VAR
	alarmP1trig: RS;		(*Триггер - защелка аварии насоса 1.*)
	alarmP2trig: RS;		(*Триггер - защелка аварии насоса 2.*)
	stopPump1Detector: F_TRIG;		(*Детектор спада сигнала (останов) насоса 1.*)
	stopPump2Detector: F_TRIG;		(*Детектор спада сигнала (останов) насоса 2.*)
	delayAfterStopP2: TOF;		(*Таймер задержки на включение
насоса 1 после останова насоса 2.*)
	delayAfterStopP1: TOF;		(*Таймер задержки на включение
насоса 2 после останова насоса 1.*)
	antiFreqStartPump1: TOF;		(*Таймер - предохранитель от частых пусков насоса 1.*)
	antiFreqStartPump2: TOF;		(*Таймер - предохранитель от частых пусков насоса 2.*)
	startPump1Trig: RS;		(*RS триггер на пуск насоса 1.*)
	startPump2Trig: RS;		(*RS триггер на пуск насоса 2.*)
	stopPump1: F_TRIG;		(*Сигнал на останов насоса 1.*)
	stopPump2: F_TRIG;		(*Сигнал на останов насоса 2.*)
END_VAR
VAR_INPUT
	startP1: BOOL;		(*Сигнал на запуск насоса 1.
Активен - пуск, неактивен - стоп.*)
	startP2: BOOL;		(*Сигнал на запуск насоса 2.
Активен - пуск, неактивен - стоп.*)
	alarmP1input: BOOL;		(*Сигнал авария от насоса 1.*)
	alarmP2input: BOOL;		(*Сигнал авария от насоса 2.*)
	stop: BOOL;		(*Сигнал на останов. Пока активен - пусков нет.
Общий на оба насоса.*)
	reset: BOOL;		(*Сброс аварий.*)
	delayTime: WORD := 300;		(*Задержка на повторный пуск в секундах.
Если ко входу ничего не подключено, то 300сек.*)
END_VAR
VAR_OUTPUT
	pump1on: BOOL;		(*Выход на запуск насоса 1.*)
	pump2on: BOOL;		(*Выход на запуск насоса 2.*)
	nextStartP1Timer: WORD;		(*Счетчик секунд до возможности повторного пуска насоса 1.*)
	nextStartP2Timer: WORD;		(*Счетчик секунд до возможности повторного пуска насоса 2.*)
	alarmP1: BOOL;		(*Статус - авария насоса 1.*)
	alarmP2: BOOL;		(*Статус - авария насоса 2.*)
END_VAR
VAR (* helpers for the ST form of the networks *)
	_t203 : TIME;
END_VAR
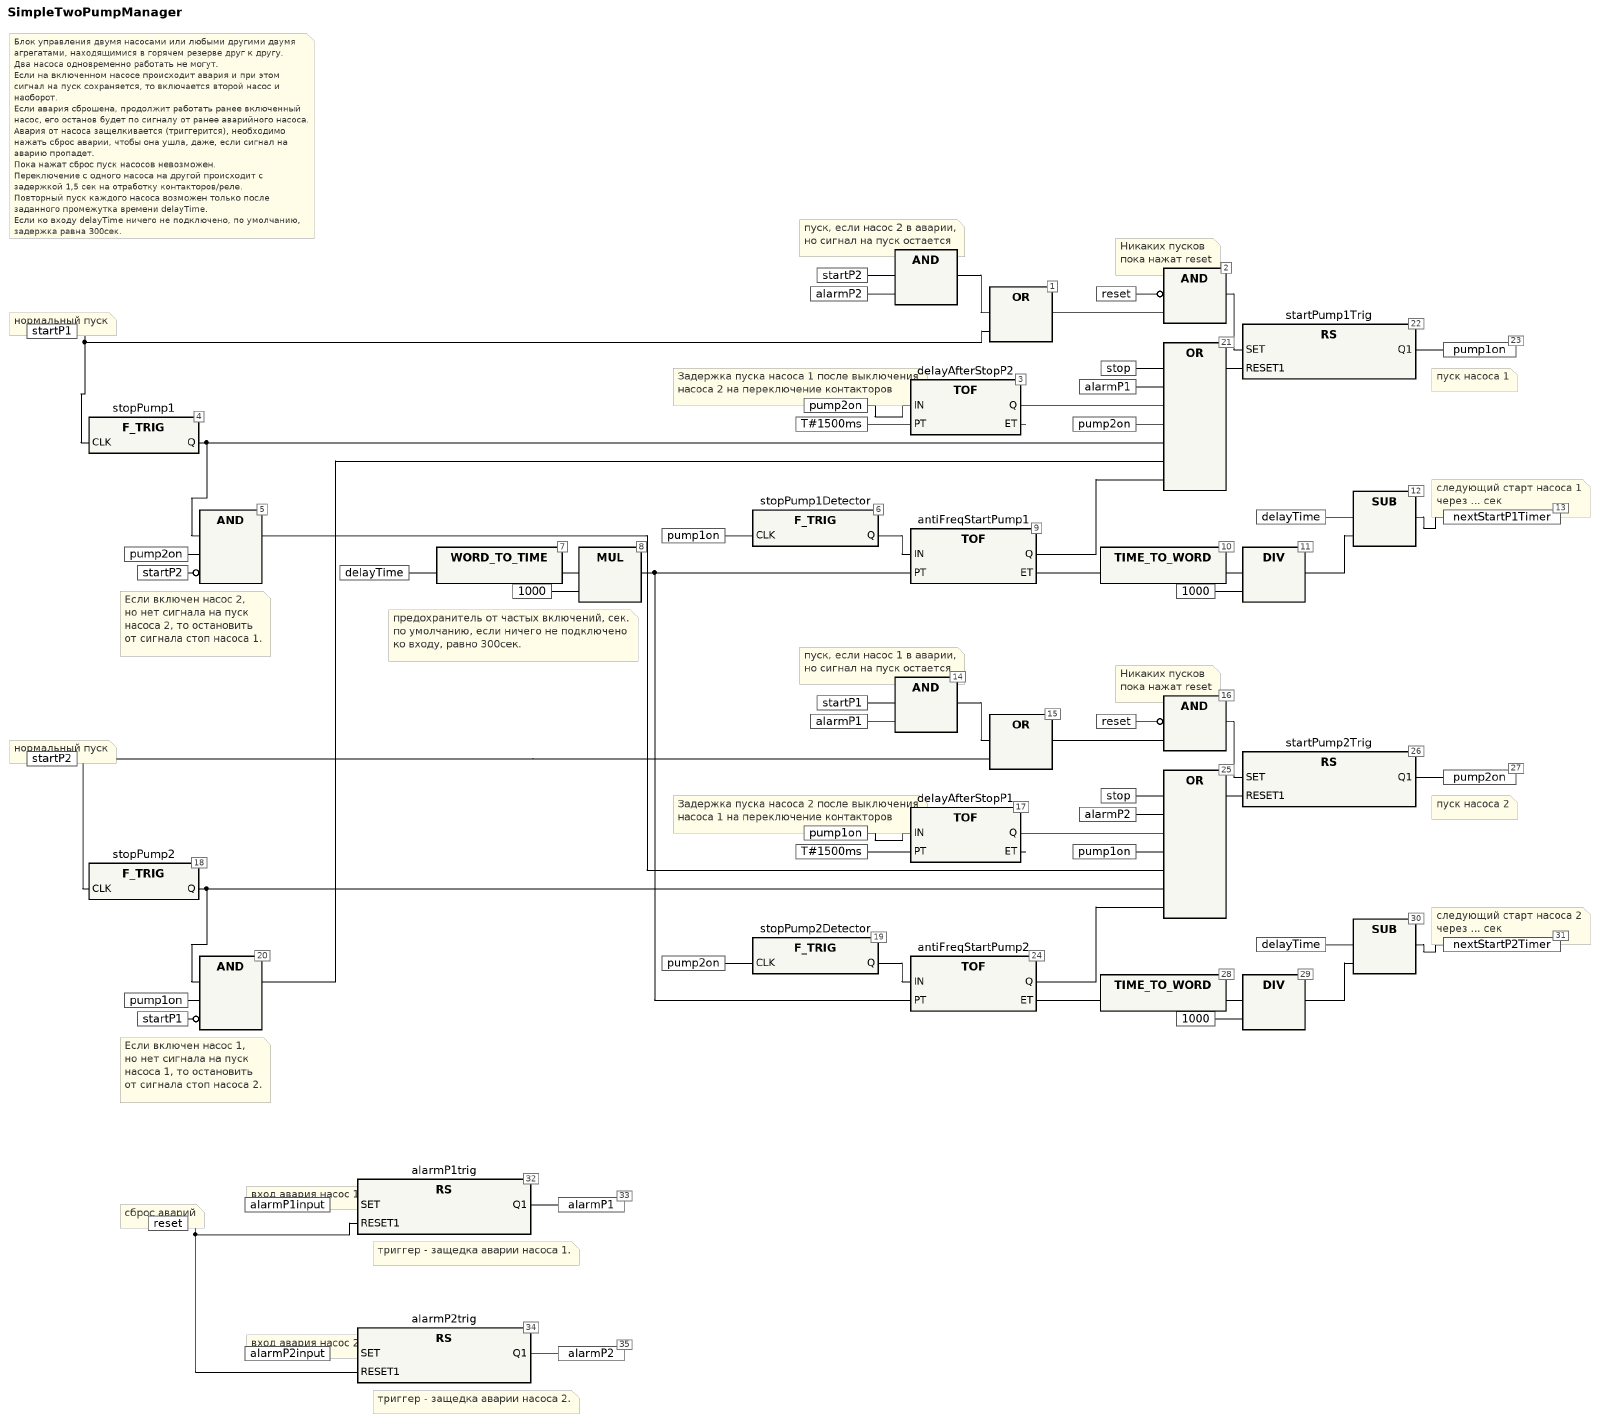
[picture p13: SimpleTwoPumpManager (CFC)]
_CFC_ (* Continuous Function Chart, elements in execution order *)
(* Задержка пуска насоса 2 после выключения / насоса 1 на переключение контакторов *)
(* cледующий старт насоса 2 / через ... сек *)
(* триггер - защедка аварии насоса 2. *)
(* cледующий старт насоса 1 / через ... сек *)
(* триггер - защедка аварии насоса 1. *)
(* предохранитель от частых включений, сек. / по умолчанию, если ничего не подключено / ко входу, равно 300сек. *)
(* пуск, если насос 1 в аварии, / но сигнал на пуск остается *)
(* нормальный пуск *)
(* пуск, если насос 2 в аварии, / но сигнал на пуск остается *)
(* нормальный пуск *)
(* Задержка пуска насоса 1 после выключения / насоса 2 на переключение контакторов *)
(* вход авария насос 1 *)
(* сброс аварий *)
(* пуск насоса 1 *)
(* вход авария насос 2 *)
(* пуск насоса 2 *)
(* Блок управления двумя насосами или любыми другими двумя агрегатами, находящимися в горячем резерве друг к другу. / Два насоса одновременно работать не могут. / Если на включенном насосе происходит авария и при этом сигнал на пуск сохраняется, то включается второй насос и наоборот. / Если авария сброшена, продолжит работать ранее включенный насос, его останов будет по сигналу от ранее аварийного насоса. / Авария от насоса защелкивается (триггерится), необходимо нажать сброс аварии, чтобы она ушла, даже, если сигнал на аварию пропадет. / Пока нажат сброс пуск насосов невозможен. / Переключение с одного насоса на другой происходит с задержкой 1,5 сек на отработку контакторов/реле. / Повторный пуск каждого насоса возможен только после заданного промежутка времени delayTime. / Если ко входу delayTime ничего не подключено, по умолчанию, задержка равна 300сек. *)
(* Никаких пусков / пока нажат reset *)
(* Никаких пусков / пока нажат reset *)
(* Если включен насос 2, / но нет сигнала на пуск / насоса 2, то остановить / от сигнала стоп насоса 1. *)
(* Если включен насос 1, / но нет сигнала на пуск / насоса 1, то остановить / от сигнала стоп насоса 2. *)
#0 AND(startP2, alarmP2)
#1 OR(#0, startP1)
#2 AND(NOT reset, #1)
#3 delayAfterStopP2:TOF(IN: pump2on, PT: T#1500ms)
#4 stopPump1:F_TRIG(CLK: startP1)
#5 AND(#4.Q, pump2on, NOT startP2)
#6 stopPump1Detector:F_TRIG(CLK: pump1on)
#7 WORD_TO_TIME(delayTime)
#8 MUL(#7, 1000)
#9 antiFreqStartPump1:TOF(IN: #6.Q, PT: #8)
#10 TIME_TO_WORD(#9.ET)
#11 DIV(#10, 1000)
#12 SUB(delayTime, #11)
#13 nextStartP1Timer <= #12
#14 AND(startP1, alarmP1)
#15 OR(#14, startP2)
#16 AND(NOT reset, #15)
#17 delayAfterStopP1:TOF(IN: pump1on, PT: T#1500ms)
#18 stopPump2:F_TRIG(CLK: startP2)
#19 stopPump2Detector:F_TRIG(CLK: pump2on)
#20 AND(#18.Q, pump1on, NOT startP1)
#21 OR(stop, alarmP1, #3.Q, pump2on, #4.Q, #20, #9.Q)
#22 startPump1Trig:RS(SET: #2, RESET1: #21)
#23 pump1on <= #22.Q1
#24 antiFreqStartPump2:TOF(IN: #19.Q, PT: #8)
#25 OR(stop, alarmP2, #17.Q, pump1on, #5, #18.Q, #24.Q)
#26 startPump2Trig:RS(SET: #16, RESET1: #25)
#27 pump2on <= #26.Q1
#28 TIME_TO_WORD(#24.ET)
#29 DIV(#28, 1000)
#30 SUB(delayTime, #29)
#31 nextStartP2Timer <= #30
#32 alarmP1trig:RS(SET: alarmP1input, RESET1: reset)
#33 alarmP1 <= #32.Q1
#34 alarmP2trig:RS(SET: alarmP2input, RESET1: reset)
#35 alarmP2 <= #34.Q1
_END_CFC_
(* the same logic as Structured Text *)
(* Задержка пуска насоса 2 после выключения / насоса 1 на переключение контакторов *)
(* cледующий старт насоса 2 / через ... сек *)
(* триггер - защедка аварии насоса 2. *)
(* cледующий старт насоса 1 / через ... сек *)
(* триггер - защедка аварии насоса 1. *)
(* предохранитель от частых включений, сек. / по умолчанию, если ничего не подключено / ко входу, равно 300сек. *)
(* пуск, если насос 1 в аварии, / но сигнал на пуск остается *)
(* нормальный пуск *)
(* пуск, если насос 2 в аварии, / но сигнал на пуск остается *)
(* нормальный пуск *)
(* Задержка пуска насоса 1 после выключения / насоса 2 на переключение контакторов *)
(* вход авария насос 1 *)
(* сброс аварий *)
(* пуск насоса 1 *)
(* вход авария насос 2 *)
(* пуск насоса 2 *)
(* Блок управления двумя насосами или любыми другими двумя агрегатами, находящимися в горячем резерве друг к другу. / Два насоса одновременно работать не могут. / Если на включенном насосе происходит авария и при этом сигнал на пуск сохраняется, то включается второй насос и наоборот. / Если авария сброшена, продолжит работать ранее включенный насос, его останов будет по сигналу от ранее аварийного насоса. / Авария от насоса защелкивается (триггерится), необходимо нажать сброс аварии, чтобы она ушла, даже, если сигнал на аварию пропадет. / Пока нажат сброс пуск насосов невозможен. / Переключение с одного насоса на другой происходит с задержкой 1,5 сек на отработку контакторов/реле. / Повторный пуск каждого насоса возможен только после заданного промежутка времени delayTime. / Если ко входу delayTime ничего не подключено, по умолчанию, задержка равна 300сек. *)
(* Никаких пусков / пока нажат reset *)
(* Никаких пусков / пока нажат reset *)
(* Если включен насос 2, / но нет сигнала на пуск / насоса 2, то остановить / от сигнала стоп насоса 1. *)
(* Если включен насос 1, / но нет сигнала на пуск / насоса 1, то остановить / от сигнала стоп насоса 2. *)
delayAfterStopP2(IN := pump2on, PT := T#1500ms);
stopPump1(CLK := startP1);
stopPump1Detector(CLK := pump1on);
_t203 := WORD_TO_TIME(delayTime) * 1000;
antiFreqStartPump1(IN := stopPump1Detector.Q, PT := _t203);
nextStartP1Timer := delayTime - (TIME_TO_WORD(antiFreqStartPump1.ET) / 1000);
delayAfterStopP1(IN := pump1on, PT := T#1500ms);
stopPump2(CLK := startP2);
stopPump2Detector(CLK := pump2on);
startPump1Trig(SET := NOT reset AND ((startP2 AND alarmP2) OR startP1), RESET1 := stop OR alarmP1 OR delayAfterStopP2.Q OR pump2on OR stopPump1.Q OR (stopPump2.Q AND pump1on AND NOT startP1) OR antiFreqStartPump1.Q);
pump1on := startPump1Trig.Q1;
antiFreqStartPump2(IN := stopPump2Detector.Q, PT := _t203);
startPump2Trig(SET := NOT reset AND ((startP1 AND alarmP1) OR startP2), RESET1 := stop OR alarmP2 OR delayAfterStopP1.Q OR pump1on OR (stopPump1.Q AND pump2on AND NOT startP2) OR stopPump2.Q OR antiFreqStartPump2.Q);
pump2on := startPump2Trig.Q1;
nextStartP2Timer := delayTime - (TIME_TO_WORD(antiFreqStartPump2.ET) / 1000);
alarmP1trig(SET := alarmP1input, RESET1 := reset);
alarmP1 := alarmP1trig.Q1;
alarmP2trig(SET := alarmP2input, RESET1 := reset);
alarmP2 := alarmP2trig.Q1;
END_FUNCTION_BLOCK

(* POU TwoPumpOneDriveManager, CFC *)
FUNCTION_BLOCK TwoPumpOneDriveManager
	VAR_INPUT
	start: BOOL;		(*Сигнал на запуск насоса согласно выбранному режиму.*)
	setPump1main: BOOL;		(*Установить режим - насос 1 = главный.
Включать импульсом.*)
	setPump2main: BOOL;		(*Установить режим - насос 2 = главный.
Включать импульсом.*)
	setByCounter: BOOL;		(*Установить режим - по количеству включений.
Включать импульсом.*)
	setByWorkTime: BOOL;		(*Установить режим - по наработке.
Включать импульсом.*)
	resetPump1counter: BOOL;		(*Сброс счетчика количества включений насоса 1.*)
	resetPump2counter: BOOL;		(*Сброс счетчика количества включений насоса 2.*)
	resetWorkTimePump1: BOOL;		(*Сброс счетчика наработки насоса 1.*)
	resetWorkTimePump2: BOOL;		(*Сброс счетчика наработки насоса 2.*)
	startPump1man: BOOL;		(*Пуск насоса 1 вручную независимо от текущего режима.*)
	startPump2man: BOOL;		(*Пуск насоса 2 вручную независимо от текущего режима.*)
	stop: BOOL;		(*Стоп обоих насосов пока вход активен.
Не стоит применять для штатного останова.*)
	resetAlarms: BOOL;		(*Сброс аварий насоса.*)
	delayRepeatedStartTime: WORD;		(*Количество секунд на задержку повторного пуска насоса.
Защита от частых включений. Если ничего не подключено = 300сек.*)
	alarmPump1input: BOOL;		(*Вход от источника сигнала об аварии насоса 1.*)
	alarmPump2input: BOOL;		(*Вход от источника сигнала об аварии насоса 2.*)
	driveAlarm: BOOL;		(*Сигнал авария от ЧРП.*)
END_VAR
VAR_OUTPUT
	regimePump1Main: BOOL;		(*Текущий режим - насос 1 = главный.*)
	regimePump2Main: BOOL;		(*Текущий режим - насос 2 = главный.*)
	regimeByCounter: BOOL;		(*Текущий режим - по количеству включений.*)
	regimeByWorkTime: BOOL;		(*Текущий режим - по наработке.*)
	counterPump1: DWORD;		(*Количество включений насоса 1.*)
	counterPump2: DWORD;		(*Количество включений насоса 2.*)
	daysPump1: WORD;		(*Количество отработанных дней насоса 1.*)
	hoursPump1: WORD;		(*Количество отработанных часов насоса 1.*)
	minutesPump1: WORD;		(*Количество отработанных минут насоса 1.*)
	secondsPump1: WORD;		(*Количество отработанных секунд насоса 1.*)
	daysPump2: WORD;		(*Количество отработанных дней насоса 2.*)
	hoursPump2: WORD;		(*Количество отработанных часов насоса 2.*)
	minutesPump2: WORD;		(*Количество отработанных минут насоса 2.*)
	secondsPump2: WORD;		(*Количество отработанных секунд насоса 2.*)
	drivePower: BOOL;		(*Сигнал на включение контактора частотного преобразователя.*)
	pump1ON: BOOL;		(*Сигнал на включение контактора насоса 1.*)
	pump2ON: BOOL;		(*Сигнал на включение контактора насоса 2.*)
	startDrive: BOOL;		(*Сигнал на запуск в частотный преобразователь.*)
	nextStartP1timer: WORD;		(*Обратный отсчет до возможности повторного пуска насоса 1.*)
	nextStartP2timer: WORD;		(*Обратный отсчет до возможности повторного пуска насоса 2.*)
	alarmPump1output: BOOL;		(*Сигнал авария насоса 1.
Триггерится, нужен сброс.*)
	alarmPump2output: BOOL;		(*Сигнал авария насоса 2.
Триггерится, нужен сброс.*)
END_VAR
VAR

	RichTwoPumpManager: RichTwoPumpManager;		(*Блок управления двумя насосами.*)
	TwoPumpOneDriveModule: TwoPumpOneDriveModule;		(*Модуль управления контакторами двух насосов и питания одного частотного преобразователя.*)
END_VAR
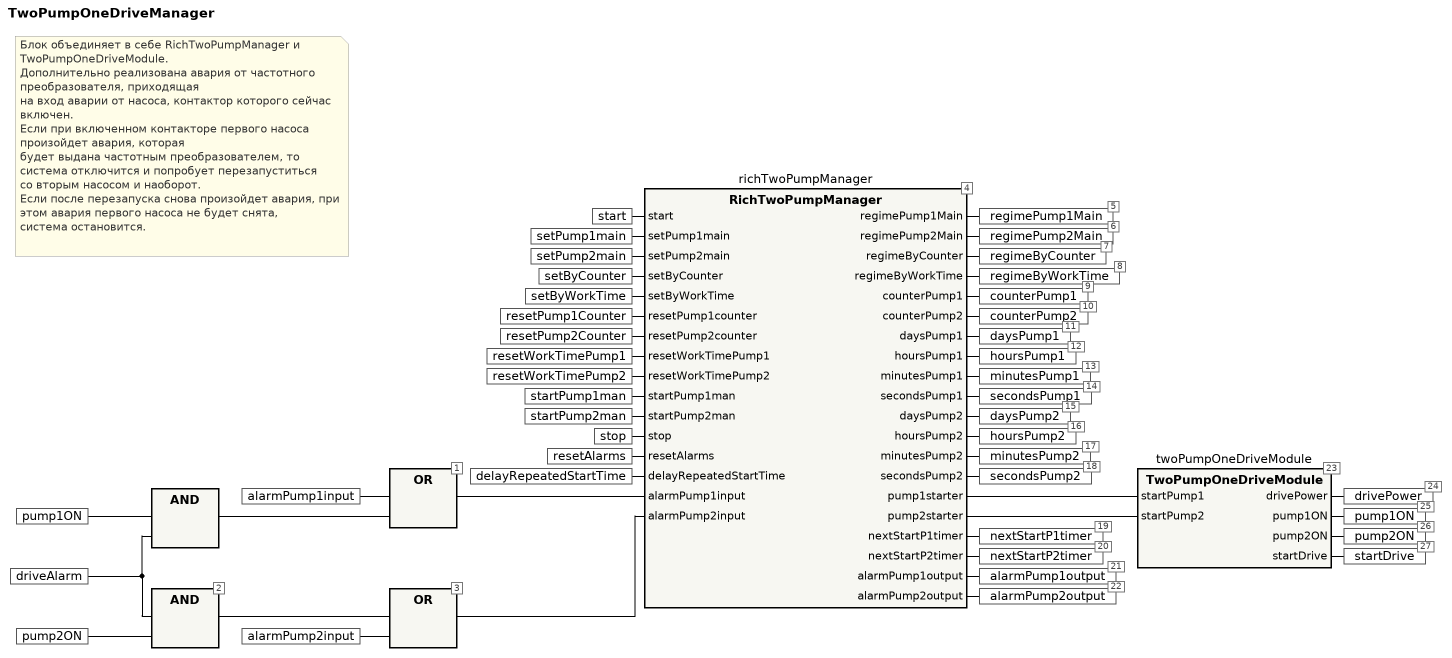
_CFC_ (* Continuous Function Chart, elements in execution order *)
(* Блок объединяет в себе RichTwoPumpManager и TwoPumpOneDriveModule. / Дополнительно реализована авария от частотного преобразователя, приходящая / на вход аварии от насоса, контактор которого сейчас включен. / Если при включенном контакторе первого насоса произойдет авария, которая / будет выдана частотным преобразователем, то система отключится и попробует перезапуститься / со вторым насосом и наоборот. / Если после перезапуска снова произойдет авария, при этом авария первого насоса не будет снята, / система остановится. *)
#0 AND(pump1ON, driveAlarm)
#1 OR(alarmPump1input, #0)
#2 AND(driveAlarm, pump2ON)
#3 OR(#2, alarmPump2input)
#4 richTwoPumpManager:RichTwoPumpManager(start: start, setPump1main: setPump1main, setPump2main: setPump2main, setByCounter: setByCounter, setByWorkTime: setByWorkTime, resetPump1counter: resetPump1Counter, resetPump2counter: resetPump2Counter, resetWorkTimePump1: resetWorkTimePump1, resetWorkTimePump2: resetWorkTimePump2, startPump1man: startPump1man, startPump2man: startPump2man, stop: stop, resetAlarms: resetAlarms, delayRepeatedStartTime: delayRepeatedStartTime, alarmPump1input: #1, alarmPump2input: #3)
#5 regimePump1Main <= #4.regimePump1Main
#6 regimePump2Main <= #4.regimePump2Main
#7 regimeByCounter <= #4.regimeByCounter
#8 regimeByWorkTime <= #4.regimeByWorkTime
#9 counterPump1 <= #4.counterPump1
#10 counterPump2 <= #4.counterPump2
#11 daysPump1 <= #4.daysPump1
#12 hoursPump1 <= #4.hoursPump1
#13 minutesPump1 <= #4.minutesPump1
#14 secondsPump1 <= #4.secondsPump1
#15 daysPump2 <= #4.daysPump2
#16 hoursPump2 <= #4.hoursPump2
#17 minutesPump2 <= #4.minutesPump2
#18 secondsPump2 <= #4.secondsPump2
#19 nextStartP1timer <= #4.nextStartP1timer
#20 nextStartP2timer <= #4.nextStartP2timer
#21 alarmPump1output <= #4.alarmPump1output
#22 alarmPump2output <= #4.alarmPump2output
#23 twoPumpOneDriveModule:TwoPumpOneDriveModule(startPump1: #4.pump1starter, startPump2: #4.pump2starter)
#24 drivePower <= #23.drivePower
#25 pump1ON <= #23.pump1ON
#26 pump2ON <= #23.pump2ON
#27 startDrive <= #23.startDrive
_END_CFC_
(* the same logic as Structured Text *)
(* Блок объединяет в себе RichTwoPumpManager и TwoPumpOneDriveModule. / Дополнительно реализована авария от частотного преобразователя, приходящая / на вход аварии от насоса, контактор которого сейчас включен. / Если при включенном контакторе первого насоса произойдет авария, которая / будет выдана частотным преобразователем, то система отключится и попробует перезапуститься / со вторым насосом и наоборот. / Если после перезапуска снова произойдет авария, при этом авария первого насоса не будет снята, / система остановится. *)
richTwoPumpManager(start := start, setPump1main := setPump1main, setPump2main := setPump2main, setByCounter := setByCounter, setByWorkTime := setByWorkTime, resetPump1counter := resetPump1Counter, resetPump2counter := resetPump2Counter, resetWorkTimePump1 := resetWorkTimePump1, resetWorkTimePump2 := resetWorkTimePump2, startPump1man := startPump1man, startPump2man := startPump2man, stop := stop, resetAlarms := resetAlarms, delayRepeatedStartTime := delayRepeatedStartTime, alarmPump1input := alarmPump1input OR (pump1ON AND driveAlarm), alarmPump2input := (driveAlarm AND pump2ON) OR alarmPump2input);
regimePump1Main := richTwoPumpManager.regimePump1Main;
regimePump2Main := richTwoPumpManager.regimePump2Main;
regimeByCounter := richTwoPumpManager.regimeByCounter;
regimeByWorkTime := richTwoPumpManager.regimeByWorkTime;
counterPump1 := richTwoPumpManager.counterPump1;
counterPump2 := richTwoPumpManager.counterPump2;
daysPump1 := richTwoPumpManager.daysPump1;
hoursPump1 := richTwoPumpManager.hoursPump1;
minutesPump1 := richTwoPumpManager.minutesPump1;
secondsPump1 := richTwoPumpManager.secondsPump1;
daysPump2 := richTwoPumpManager.daysPump2;
hoursPump2 := richTwoPumpManager.hoursPump2;
minutesPump2 := richTwoPumpManager.minutesPump2;
secondsPump2 := richTwoPumpManager.secondsPump2;
nextStartP1timer := richTwoPumpManager.nextStartP1timer;
nextStartP2timer := richTwoPumpManager.nextStartP2timer;
alarmPump1output := richTwoPumpManager.alarmPump1output;
alarmPump2output := richTwoPumpManager.alarmPump2output;
twoPumpOneDriveModule(startPump1 := richTwoPumpManager.pump1starter, startPump2 := richTwoPumpManager.pump2starter);
drivePower := twoPumpOneDriveModule.drivePower;
pump1ON := twoPumpOneDriveModule.pump1ON;
pump2ON := twoPumpOneDriveModule.pump2ON;
startDrive := twoPumpOneDriveModule.startDrive;
END_FUNCTION_BLOCK

(* POU TwoPumpOneDriveModule, CFC *)
FUNCTION_BLOCK TwoPumpOneDriveModule
VAR_INPUT
	startPump1: BOOL;		(*Входящий сигнал на запуск первого насоса.*)
	startPump2: BOOL;		(*Входящий сигнал на запуск второго насоса.*)
END_VAR
VAR_OUTPUT
	drivePower: BOOL;		(*Выход управления контактором питания ЧРП.*)
	pump1ON: BOOL;		(*Выход управления контактором питания насоса 1.*)
	pump2ON: BOOL;		(*Выход управления контактором питания насоса 2.*)
	startDrive: BOOL;		(*Сигнал пуск в ЧРП.*)
END_VAR
VAR
	pump1Off: BOOL;		(*Сигнал на отключение контактора насоса 1.*)
	pump2Off: BOOL;		(*Сигнал на отключение контактора насоса 2.*)
	startP1trig: R_TRIG;		(*Триггер переднего фронта сигнала на запуск насоса 1.*)
	startP2trig: R_TRIG;		(*Триггер переднего фронта сигнала на запуск насоса 2.*)
	ifP1on: IfBOOL;		(*Блок отправляет сигнал на запуск насоса 1 по одной
			из двух веток в зависимости от состояния ключа.*)
	ifP2on: IfBOOL;		(*Блок отправляет сигнал на запуск насоса 2 по одной
			из двух веток в зависимости от состояния ключа.*)
	startDriveDelay: TON;		(*Блок задержки подачи сигнала на включение ЧРП.*)
	stopDriveTrig: F_TRIG;		(*Триггер спада сигнала на включение насоса 1 или 2 для
			снятия сигнала пуск в ЧРП.*)
	p1ONdelay: TON;		(*Задержка на включение контактора насоса 1.*)
	p2ONdelay: TON;		(*Задержка на включение контактора насоса 2.*)
	startDriveTrig: RS;		(*RS триггер сигнала пуск в ЧРП.*)
	p1powerTrig: RS;		(*RS триггер включения контактора насоса 1.*)
	p2powerTrig: RS;		(*RS триггер включения контактора насоса 2.*)
	offP1delayTrig: RS;		(*RS триггер сигнала на отключение контактора насоса 1.*)
	offP2delayTrig: RS;		(*RS триггер сигнала на отключение контактора насоса 2.*)
	offPowerDelay: TOF;		(*Блок управления временем выключения контактора питания ЧРП.*)
	offP2delay: TON;		(*Задержка выключения контактора насоса 1.*)
	offP1delay: TON;		(*Задержка выключения контактора насоса 2.*)
	fastStart: BOOL;		(*Быстрый сигнал на пуск в ЧРП, если не надо переключать
			контакторы.*)
END_VAR
VAR (* helpers for the ST form of the networks *)
	_t160 : BOOL;
END_VAR
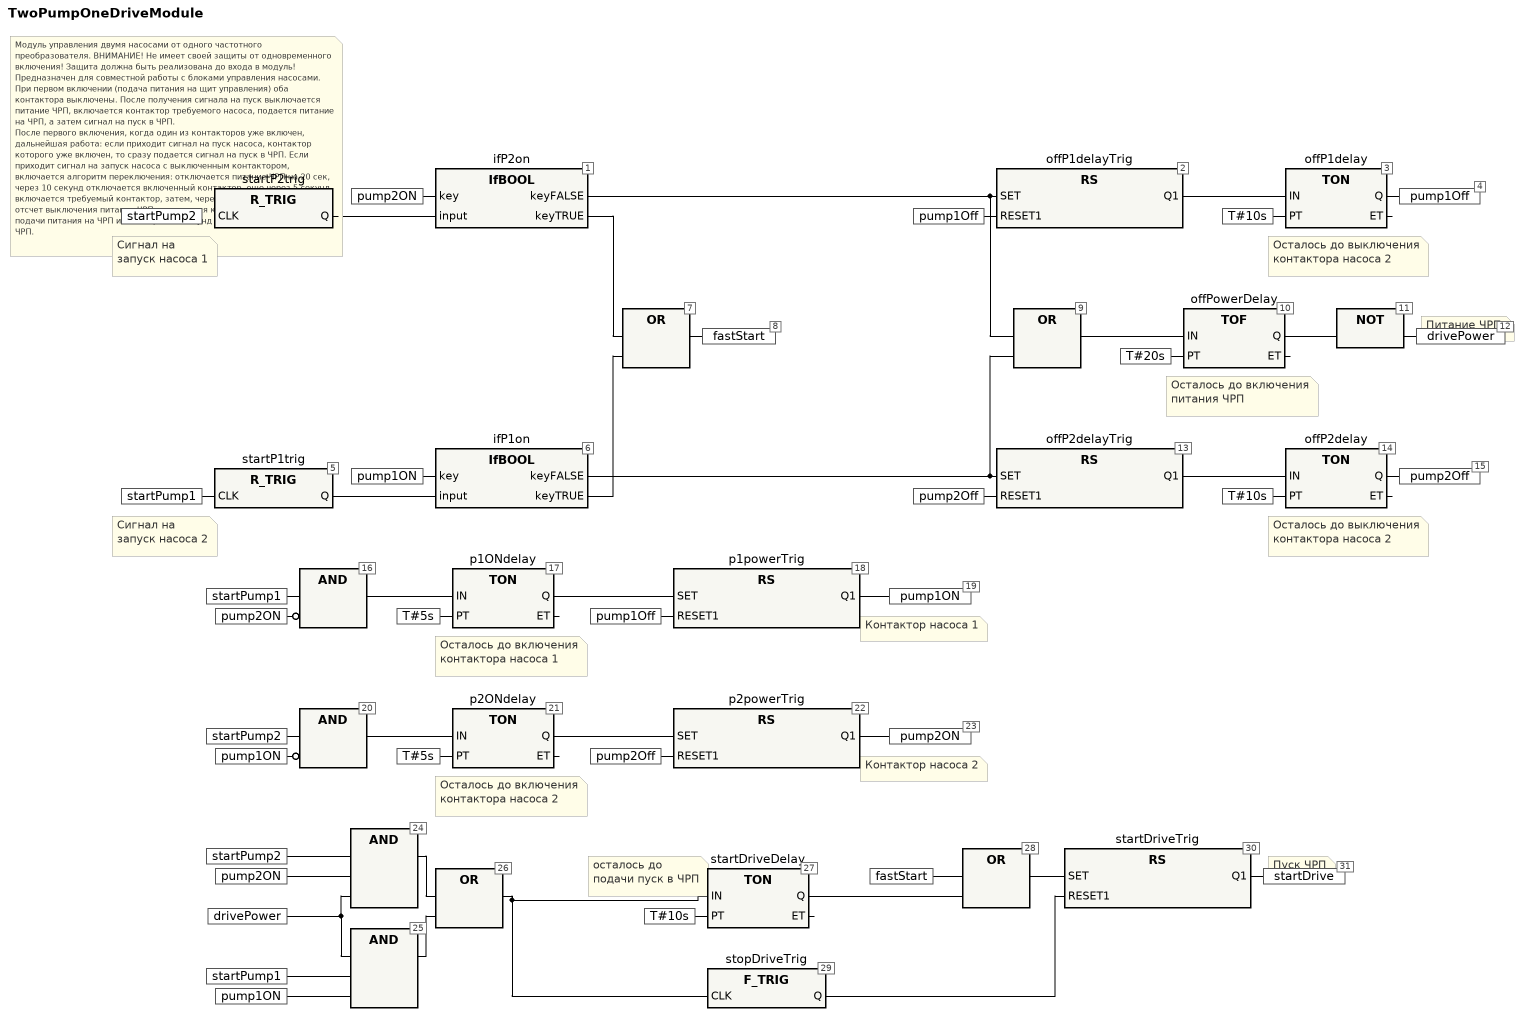
_CFC_ (* Continuous Function Chart, elements in execution order *)
(* Модуль управления двумя насосами от одного частотного преобразователя. ВНИМАНИЕ! Не имеет своей защиты от одновременного включения! Защита должна быть реализована до входа в модуль! Предназначен для совместной работы с блоками управления насосами. / При первом включении (подача питания на щит управления) оба контактора выключены. После получения сигнала на пуск выключается питание ЧРП, включается контактор требуемого насоса, подается питание на ЧРП, а затем сигнал на пуск в ЧРП. / После первого включения, когда один из контакторов уже включен, дальнейшая работа: если приходит сигнал на пуск насоса, контактор которого уже включен, то сразу подается сигнал на пуск в ЧРП. Если приходит сигнал на запуск насоса с выключенным контактором, / включается алгоритм переключения: отключается питание ЧРП на 20 сек, через 10 секунд отключается включенный контактор, еще через 5 секунд включается требуемый контактор, затем, через 5 секунд, заканчивается отсчет выключения питания ЧРП, включается контактор / подачи питания на ЧРП и еще через 10 секунд подается питание на пуск в ЧРП. *)
(* Сигнал на / запуск насоса 2 *)
(* Сигнал на / запуск насоса 1 *)
(* Контактор насоса 1 *)
(* Осталось до включения / контактора насоса 1 *)
(* Контактор насоса 2 *)
(* Осталось до выключения / контактора насоса 2 *)
(* Осталось до включения / питания ЧРП *)
(* Питание ЧРП. *)
(* Осталось до включения / контактора насоса 2 *)
(* Осталось до выключения / контактора насоса 2 *)
(* осталось до / подачи пуск в ЧРП *)
(* Пуск ЧРП *)
#0 startP2trig:R_TRIG(CLK: startPump2)
#1 ifP2on:IfBOOL(key: pump2ON, input: #0.Q)
#2 offP1delayTrig:RS(SET: #1.keyFALSE, RESET1: pump1Off)
#3 offP1delay:TON(IN: #2.Q1, PT: T#10s)
#4 pump1Off <= #3.Q
#5 startP1trig:R_TRIG(CLK: startPump1)
#6 ifP1on:IfBOOL(key: pump1ON, input: #5.Q)
#7 OR(#1.keyTRUE, #6.keyTRUE)
#8 fastStart <= #7
#9 OR(#1.keyFALSE, #6.keyFALSE)
#10 offPowerDelay:TOF(IN: #9, PT: T#20s)
#11 NOT(#10.Q)
#12 drivePower <= #11
#13 offP2delayTrig:RS(SET: #6.keyFALSE, RESET1: pump2Off)
#14 offP2delay:TON(IN: #13.Q1, PT: T#10s)
#15 pump2Off <= #14.Q
#16 AND(startPump1, NOT pump2ON)
#17 p1ONdelay:TON(IN: #16, PT: T#5s)
#18 p1powerTrig:RS(SET: #17.Q, RESET1: pump1Off)
#19 pump1ON <= #18.Q1
#20 AND(startPump2, NOT pump1ON)
#21 p2ONdelay:TON(IN: #20, PT: T#5s)
#22 p2powerTrig:RS(SET: #21.Q, RESET1: pump2Off)
#23 pump2ON <= #22.Q1
#24 AND(startPump2, pump2ON, drivePower)
#25 AND(drivePower, startPump1, pump1ON)
#26 OR(#24, #25)
#27 startDriveDelay:TON(IN: #26, PT: T#10s)
#28 OR(fastStart, #27.Q)
#29 stopDriveTrig:F_TRIG(CLK: #26)
#30 startDriveTrig:RS(SET: #28, RESET1: #29.Q)
#31 startDrive <= #30.Q1
_END_CFC_
(* the same logic as Structured Text *)
(* Модуль управления двумя насосами от одного частотного преобразователя. ВНИМАНИЕ! Не имеет своей защиты от одновременного включения! Защита должна быть реализована до входа в модуль! Предназначен для совместной работы с блоками управления насосами. / При первом включении (подача питания на щит управления) оба контактора выключены. После получения сигнала на пуск выключается питание ЧРП, включается контактор требуемого насоса, подается питание на ЧРП, а затем сигнал на пуск в ЧРП. / После первого включения, когда один из контакторов уже включен, дальнейшая работа: если приходит сигнал на пуск насоса, контактор которого уже включен, то сразу подается сигнал на пуск в ЧРП. Если приходит сигнал на запуск насоса с выключенным контактором, / включается алгоритм переключения: отключается питание ЧРП на 20 сек, через 10 секунд отключается включенный контактор, еще через 5 секунд включается требуемый контактор, затем, через 5 секунд, заканчивается отсчет выключения питания ЧРП, включается контактор / подачи питания на ЧРП и еще через 10 секунд подается питание на пуск в ЧРП. *)
(* Сигнал на / запуск насоса 2 *)
(* Сигнал на / запуск насоса 1 *)
(* Контактор насоса 1 *)
(* Осталось до включения / контактора насоса 1 *)
(* Контактор насоса 2 *)
(* Осталось до выключения / контактора насоса 2 *)
(* Осталось до включения / питания ЧРП *)
(* Питание ЧРП. *)
(* Осталось до включения / контактора насоса 2 *)
(* Осталось до выключения / контактора насоса 2 *)
(* осталось до / подачи пуск в ЧРП *)
(* Пуск ЧРП *)
startP2trig(CLK := startPump2);
ifP2on(key := pump2ON, input := startP2trig.Q);
offP1delayTrig(SET := ifP2on.keyFALSE, RESET1 := pump1Off);
offP1delay(IN := offP1delayTrig.Q1, PT := T#10s);
pump1Off := offP1delay.Q;
startP1trig(CLK := startPump1);
ifP1on(key := pump1ON, input := startP1trig.Q);
fastStart := ifP2on.keyTRUE OR ifP1on.keyTRUE;
offPowerDelay(IN := ifP2on.keyFALSE OR ifP1on.keyFALSE, PT := T#20s);
drivePower := NOT offPowerDelay.Q;
offP2delayTrig(SET := ifP1on.keyFALSE, RESET1 := pump2Off);
offP2delay(IN := offP2delayTrig.Q1, PT := T#10s);
pump2Off := offP2delay.Q;
p1ONdelay(IN := startPump1 AND NOT pump2ON, PT := T#5s);
p1powerTrig(SET := p1ONdelay.Q, RESET1 := pump1Off);
pump1ON := p1powerTrig.Q1;
p2ONdelay(IN := startPump2 AND NOT pump1ON, PT := T#5s);
p2powerTrig(SET := p2ONdelay.Q, RESET1 := pump2Off);
pump2ON := p2powerTrig.Q1;
_t160 := (startPump2 AND pump2ON AND drivePower) OR (drivePower AND startPump1 AND pump1ON);
startDriveDelay(IN := _t160, PT := T#10s);
stopDriveTrig(CLK := _t160);
startDriveTrig(SET := fastStart OR startDriveDelay.Q, RESET1 := stopDriveTrig.Q);
startDrive := startDriveTrig.Q1;
END_FUNCTION_BLOCK
